{region '#Template'}
	{attribute 'Version' := '1.3.2.0'}
	{attribute 'Tags' := '"LCID": "1031", "Text": "AC, Aggregates, pre-heater"'}
	{attribute 'Tags' := '"LCID": "1033", "Text": "AC, Aggregates, pre-heater"'}
	{attribute 'Using' := '"Type": "Template", "URI": "BA2_Param"'}
	{attribute 'Using' := '"Type": "Template", "URI": "EC_AMEV"'}
	{attribute 'Description' := '"LCID": "1031", "Text": "Aggregat Vorerhitzer"'}
	{attribute 'Description' := '"LCID": "1033", "Text": "Aggregate pre-heater"'}
{endregion}
FUNCTION_BLOCK FB_BA_AC_PreHtr EXTENDS FB_BA_AggregateB
VAR_INPUT
	fSpTSuA					: REAL;
	fTSuA					: REAL;
	bDehumf					: BOOL;
	bMixADmpAvail			: BOOL;
	fTWth					: REAL;
	bTWthLowLimit			: BOOL;
	bResetDehumf    		: BOOL;	
END_VAR
VAR_OUTPUT
	bCmd					: BOOL;
	fPresentValue			: REAL;			
	bFrost					: BOOL;
	bPreRinse				: BOOL;
	bActiveSeqCtrl			: BOOL;	
END_VAR
VAR_INPUT CONSTANT PERSISTENT
	{attribute 'parameterCategory' := 'Behaviour'}
	fHysPuOn : REAL := 5.0;
	{attribute 'parameterCategory' := 'Behaviour'}
	fHysPuOff : REAL := 1.0;
END_VAR
VAR_INPUT CONSTANT
	TFl						: FB_BA_SensorAnalog_IO;												
	TRt						: FB_BA_SensorAnalog_IO;			
	ProcessPreRinse			: FB_BA_Process;		
	TSuACtrl				: FB_BA_AC_PreHtrTSuACtrl;
	TRtCtrl					: FB_BA_AC_TRtCtrl;	
	TFrost					: FB_BA_SensorAnalog_IO;																	
	TFrostPrtcCtrlAir		: FB_BA_PID_Sp;
	FrostThermostat			: FB_BA_SensorBinary_IO;
	Vlv						: FB_BA_Vlv;
	Pu						: FB_BA_Pu1st; 							
END_VAR
VAR
	HysPu					: FB_BA_Swi2P;
	rsForceSeq				: RS;
END_VAR
VAR // added by the converter: edge detectors and wires of the graphical bodies
    _w1 : ANY;
    _w2 : BOOL;
END_VAR

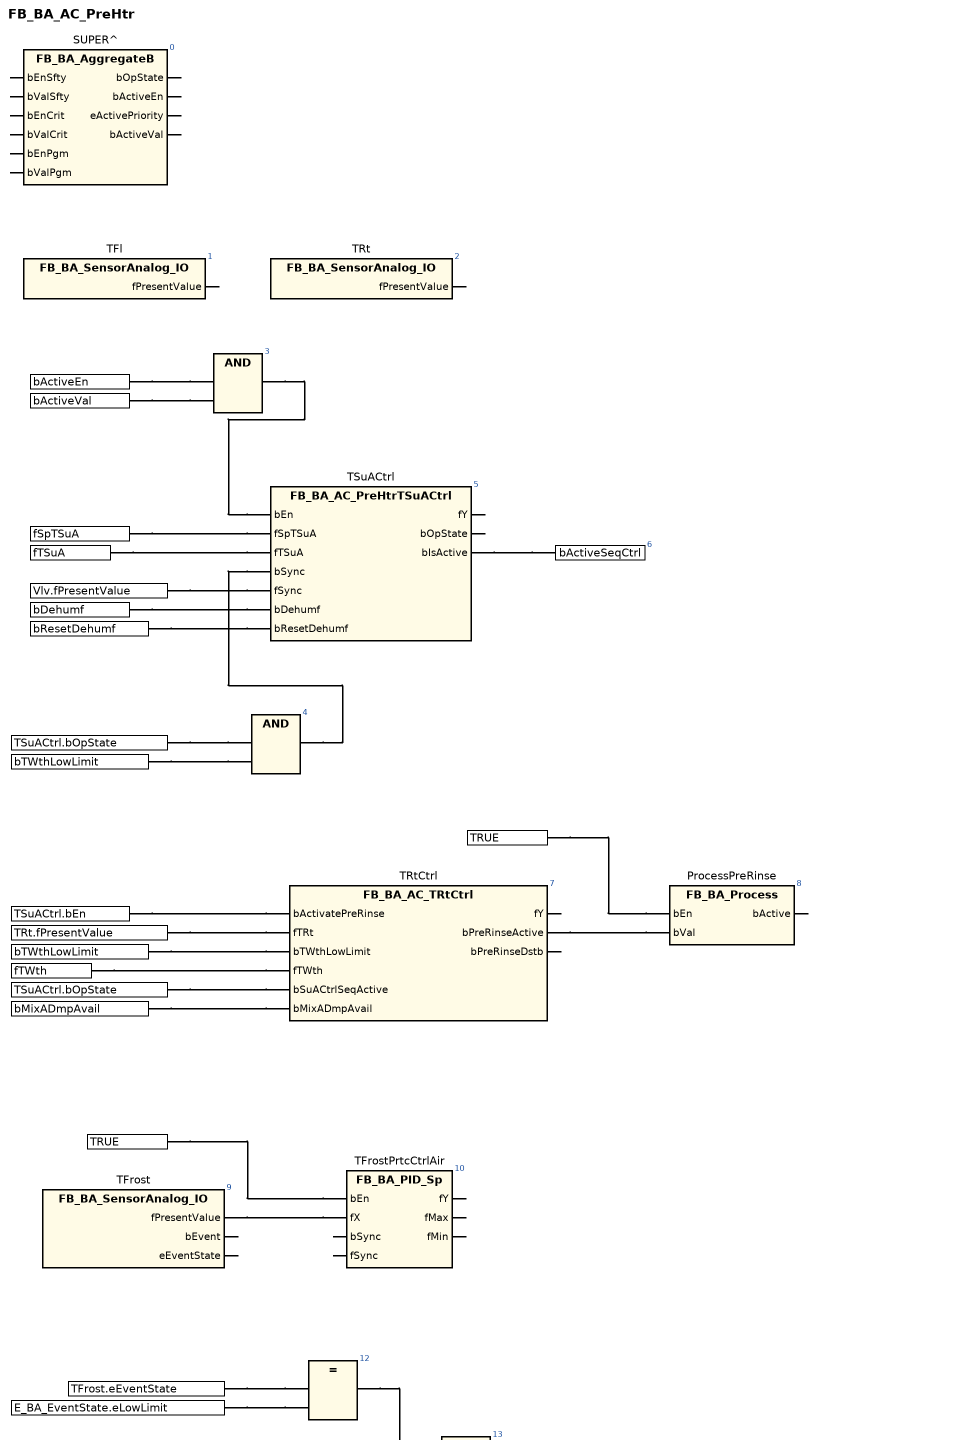
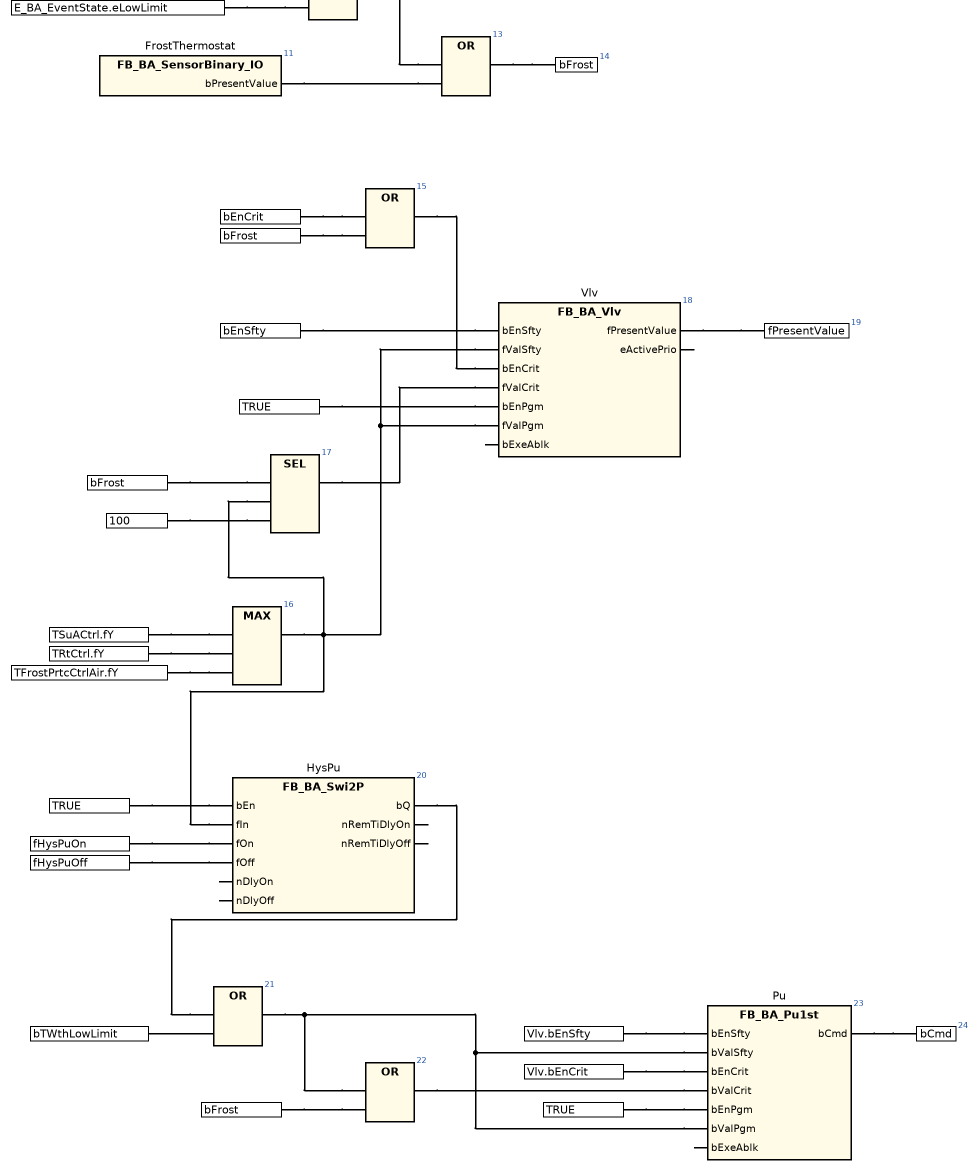
SUPER^(); // FB_BA_AggregateB
TFl(); // FB_BA_SensorAnalog_IO
TRt(); // FB_BA_SensorAnalog_IO
TSuACtrl(
    bEn := bActiveEn AND bActiveVal,
    fSpTSuA := fSpTSuA,
    fTSuA := fTSuA,
    bSync := TSuACtrl.bOpState AND bTWthLowLimit,
    fSync := Vlv.fPresentValue,
    bDehumf := bDehumf,
    bResetDehumf := bResetDehumf); // FB_BA_AC_PreHtrTSuACtrl
bActiveSeqCtrl := TSuACtrl.bIsActive;
TRtCtrl(
    bActivatePreRinse := TSuACtrl.bEn,
    fTRt := TRt.fPresentValue,
    bTWthLowLimit := bTWthLowLimit,
    fTWth := fTWth,
    bSuACtrlSeqActive := TSuACtrl.bOpState,
    bMixADmpAvail := bMixADmpAvail); // FB_BA_AC_TRtCtrl
ProcessPreRinse(bEn := TRUE, bVal := TRtCtrl.bPreRinseActive); // FB_BA_Process
TFrost(); // FB_BA_SensorAnalog_IO
TFrostPrtcCtrlAir(bEn := TRUE, fX := TFrost.fPresentValue); // FB_BA_PID_Sp
FrostThermostat(); // FB_BA_SensorBinary_IO
bFrost := TFrost.eEventState = E_BA_EventState.eLowLimit OR FrostThermostat.bPresentValue;
_w1 := MAX(TSuACtrl.fY, TRtCtrl.fY, TFrostPrtcCtrlAir.fY);
Vlv(
    bEnSfty := bEnSfty,
    fValSfty := _w1,
    bEnCrit := bEnCrit OR bFrost,
    fValCrit := SEL(bFrost, _w1, 100),
    bEnPgm := TRUE,
    fValPgm := _w1); // FB_BA_Vlv
fPresentValue := Vlv.fPresentValue;
HysPu(bEn := TRUE, fIn := _w1, fOn := fHysPuOn, fOff := fHysPuOff); // FB_BA_Swi2P
_w2 := HysPu.bQ OR bTWthLowLimit;
Pu(
    bEnSfty := Vlv.bEnSfty,
    bValSfty := _w2,
    bEnCrit := Vlv.bEnCrit,
    bValCrit := _w2 OR bFrost,
    bEnPgm := TRUE,
    bValPgm := _w2); // FB_BA_Pu1st
bCmd := Pu.bCmd;

METHOD FB_init : BOOL
VAR_INPUT
	bInitRetains : BOOL; // if TRUE, the retain variables are initialized (warm start / cold start)
	bInCopyCode : BOOL;  // if TRUE, the instance afterwards gets moved into the copy code (online change)
END_VAR
TFl.iParent										:= THIS^;		
TFl.iLabel 										:= LblCmpAC.PreHtr_TFl;	
TFl.sObjectName									:= '{Idx=11}';
TFl.eDPADMode									:= E_BA_DPADMode.eInclude;
TFl.MV.eUnit									:= E_BA_Unit.eTemperature_DegreesCelsius;
TFl.MV.fResolution 								:= 0.01;
TFl.MV.fScaleOffset 							:= 0; 
TFl.MV.bEventDetectionEnable					:= TRUE;
TFl.MV.eEnPlantLock								:= E_BA_LockPriority.eNoLock;
                            					                            					
TRt.iParent										:= THIS^;		
TRt.iLabel 										:= LblCmpAC.PreHtr_TRt;	
TRt.sObjectName									:= '{Idx=11}';
TRt.eDPADMode									:= E_BA_DPADMode.eInclude;
TRt.MV.eUnit									:= E_BA_Unit.eTemperature_DegreesCelsius;
TRt.MV.fResolution 								:= 0.01;
TRt.MV.fScaleOffset 							:= 0;  
TRt.MV.bEventDetectionEnable					:= TRUE;
TRt.MV.eEnPlantLock								:= E_BA_LockPriority.eMedium;

ProcessPreRinse.Parent 							:= THIS^;
ProcessPreRinse.Label							:= LblCmpAC.PreHtr_ProcessPreRinse;

TSuACtrl.iParent								:= THIS^;	
TSuACtrl.iLabel									:= LblCmpAC.PreHtr_TSuACtrl;
TSuACtrl.sObjectName							:= '{Idx=11}';										 
TSuACtrl.eDPADMode								:= E_BA_DPADMode.eInclude;								

TRtCtrl.iParent									:= THIS^;
TRtCtrl.iLabel									:= LblCmpAC.PreHtr_TRtCtrl;
TRtCtrl.sObjectName								:= '{Idx=12}';										 
TRtCtrl.eDPADMode								:= E_BA_DPADMode.eInclude;								
TRtCtrl.PreRinseDst.bEventDetectionEnable	:= TRUE;
TRtCtrl.PreRinseDst.eEnPlantLock				:= E_BA_LockPriority.eNoLock;
	                                				
TFrost.iParent									:= THIS^;		
TFrost.iLabel 									:= LblCmpAC.PreHtr_TFrost;	
TFrost.sObjectName								:= '{Idx=11}';
TFrost.eDPADMode								:= E_BA_DPADMode.eInclude;
TFrost.MV.eUnit									:= E_BA_Unit.eTemperature_DegreesCelsius;
TFrost.MV.fResolution 							:= 0.0004577776;
TFrost.MV.fScaleOffset 							:= 0;  
TFrost.MV.bEventDetectionEnable				:= TRUE;
TFrost.MV.eEnPlantLock							:= E_BA_LockPriority.eMedium;

TFrostPrtcCtrlAir.iParent						:= THIS^;	
TFrostPrtcCtrlAir.iLabel						:= LblCmpAC.PreHtr_TFrostPrtcCtrlAir;
TFrostPrtcCtrlAir.sObjectName					:= '{Idx=13}';										 
TFrostPrtcCtrlAir.eDPADMode						:= E_BA_DPADMode.eInclude;
TFrostPrtcCtrlAir.Sp.fValueRm 					:= 5.0;
TFrostPrtcCtrlAir.Ctrl.fProportionalConstant	:= 5;
TFrostPrtcCtrlAir.Ctrl.fIntegralConstant		:= 60;	
TFrostPrtcCtrlAir.Ctrl.eActionRm				:= E_BA_Action.eReverse;

FrostThermostat.iParent							:= THIS^;
FrostThermostat.iLabel							:= LblCmpAC.PreHtr_FrostThermostat;												 										 
FrostThermostat.sObjectName						:= '{Idx=11}';
FrostThermostat.eDPADMode						:= E_BA_DPADMode.eInclude;
FrostThermostat.Input.iLabel					:= LblFunctions_OperationalMessage;	
FrostThermostat.Input.sObjectName				:= '{Idx=01}';	
FrostThermostat.Input.ePolarity					:= E_BA_Polarity.eReverse;
FrostThermostat.Input.sActiveText 				:= txtEvent_Triggered;
FrostThermostat.Input.sInactiveText 			:= txtEvent_Normal;
FrostThermostat.Input.nEventClassID				:= EC_ID.NC30;
FrostThermostat.Input.aEventTransitionText[1]	:= txtEvent_Triggered;
FrostThermostat.Input.aEventTransitionText[2]	:= txtEvent_Error;
FrostThermostat.Input.aEventTransitionText[3]	:= txtEvent_Normal;
FrostThermostat.Input.bEventDetectionEnable		:= TRUE;
FrostThermostat.Input.eEnPlantLock				:= E_BA_LockPriority.eMedium;	

Vlv.iParent										:= THIS^;
Vlv.iLabel										:= LblCmpAC.PreHtr_Vlv;
Vlv.sObjectName									:= '{Idx=11}';										 
Vlv.eDPADMode									:= E_BA_DPADMode.eInclude;								
                            					
Pu.iParent										:= THIS^;
Pu.iLabel										:= LblCmpAC.PreHtr_Pu;
Pu.sObjectName									:= '{Idx=11}';										 
Pu.eDPADMode									:= E_BA_DPADMode.eInclude;
Pu.Dst.bEventDetectionEnable					:= TRUE;
Pu.Dst.eEnPlantLock								:= E_BA_LockPriority.eMedium;
END_METHOD

END_FUNCTION_BLOCK

(* stored: Version 1.1.0.1, ProductVersion 3.1.4024.9
   POU FB_BA_AC_PreHtr: Id {e9359802-b996-4d44-b348-d6888cea29c4}, SpecialFunc None
   Method FB_init: Id {b1a09a06-2335-4c6f-a86c-3c5cf1e0fcf6} *)
